// TIA Portal V19 export
VAR_GLOBAL   // PLC tag table "MotionTags"
END_VAR
